		fbUnitTest.addString('<?xml version="1.0" ?>');
		fbUnitTest.addCrlf();

		fbUnitTest.addString('<testsuites>');
		fbUnitTest.addCrlf();

		pActTestSuite := getFirstTestSuite();

		WHILE (pActTestSuite <> 0) DO

			u16TestSuitIdx := u16TestSuitIdx+1;

			fbUnitTest.addString('<testsuite');
			fbUnitTest.addString(' name="');
			fbUnitTest.addString(pActTestSuite^.getId());
			fbUnitTest.addString('" tests="');
			u32Temp := pActTestSuite^.getNoOfTests();
			fbUnitTest.addValue(u32Temp);
			fbUnitTest.addString('" disabled="');
			u32Temp := 0;
			fbUnitTest.addValue(u32Temp);
			fbUnitTest.addString('" errors="');
			fbUnitTest.addValue(u32Temp);
			fbUnitTest.addString('" failures="');
			u32Temp := pActTestSuite^.getFailed();
			fbUnitTest.addValue(u32Temp);
			fbUnitTest.addString('" hostname="');
			fbUnitTest.addString('" id="');
			fbUnitTest.addvalue(u16TestSuitIdx);
			fbUnitTest.addString('" package="');
			fbUnitTest.addString(pActTestSuite^.getPath());
			fbUnitTest.addString('">');
			fbUnitTest.addCrlf();

			pTestCase := pActTestSuite^.getFirstTestCase();

			WHILE (pTestCase <> 0) DO

				fbUnitTest.addString('<testcase');
				fbUnitTest.addString(' name="');
				fbUnitTest.addString(pTestCase^.getId());
				fbUnitTest.addString('" assertions="');
				u32Temp := pTestCase^.getFailed() + pTestCase^.getPassed();
				fbUnitTest.addValue(u32Temp);
				fbUnitTest.addString('" classname="');
				fbUnitTest.addString(pTestCase^.getPath());
				fbUnitTest.addString(pTestCase^.getClassName());
				fbUnitTest.addString('" time="');
				u32Temp := pTestCase^.getTime();
				fbUnitTest.addTimeMs(u32Temp);
				fbUnitTest.addString('">');
				fbUnitTest.addCrlf();

				CASE pTestCase^.o_eResult OF

				EResult_t.eStatePassed :

					fbUnitTest.addString('<passed/>');

				EResult_t.eStateFailed, 
				EResult_t.eStateFailedFatal :
			
					fbUnitTest.addString('<failure');
					fbUnitTest.addString(' message="');
					fbUnitTest.addString(pTestCase^.getMessage());
					fbUnitTest.addString('"/>');
					
				EResult_t.eStateSkipped:

					fbUnitTest.addString('<skipped/>');

				END_CASE;
				
				fbUnitTest.addCrlf();	

				fbUnitTest.addString('</testcase>');
				fbUnitTest.addCrlf();		

				pTestCase := pActTestSuite^.getNextTestCase();
		
			END_WHILE

			fbUnitTest.addString('</testsuite>');
			fbUnitTest.addCrlf();	

			pActTestSuite := getNextTestSuite();

		END_WHILE

		fbUnitTest.addString('</testsuites>');
		fbUnitTest.addCrlf();

		u16ReportState := 22;

	22:
		IF fbUnitTest.o_bOpen  = TRUE AND 
		   fbUnitTest.o_bEmpty = TRUE THEN
			fbUnitTest.close();
		END_IF;

		IF fbUnitTest.o_bOpen  = FALSE THEN
			createReport 	:= ERetCode_t.eRetDone;
		END_IF;

// +++++++++++++++++++++++++++++++++++++++++++++++++++++++++++
//
//
// 
// +++++++++++++++++++++++++++++++++++++++++++++++++++++++++++
	100:

		IF pTestReport <> 0 THEN
			
			createReport := pTestReport^.create();		
			
		ELSE

			createReport := ERetCode_t.eRetDone;

		END_IF;

	ELSE
		createReport := ERetCode_t.eRetFailed;
	END_CASE;

	IF createReport = ERetCode_t.eRetDone THEN
		u16ReportState := 0;
	END_IF;
















(**)
END_METHOD

(******************************************************************************
Baustein: PRG_UnitTestLib.getFirstTestSuite
Spezifikation: doc/Spezifikation.pdf, Kap. x.y.z
-------------------------------------------------------------------------------
erstellt:
von:
Geändert:
von:
-------------------------------------------------------------------------------
Beschreibung
Diese Methode

-------------------------------------------------------------------------------
Input
-

Output
-
******************************************************************************)
{attribute 'hide'} 
METHOD PRIVATE getFirstTestSuite : TestSuiteHandle_t
VAR_INPUT
END_VAR

	u16Index := 0;
	getFirstTestSuite := a_pTestSuite[0];
END_METHOD

(******************************************************************************
Baustein: PRG_UnitTestLib.getNextTestSuite
Spezifikation: doc/Spezifikation.pdf, Kap. x.y.z
-------------------------------------------------------------------------------
erstellt:
von:
Geändert:
von:
-------------------------------------------------------------------------------
Beschreibung
Diese Methode

-------------------------------------------------------------------------------
Input
-

Output
-
******************************************************************************)
{attribute 'hide'} 
METHOD PRIVATE getNextTestSuite : TestSuiteHandle_t
VAR_INPUT
END_VAR

	getNextTestSuite := 0;
	u16Index 		 := u16Index + 1;

	IF u16Index < u16TestSuites THEN
		getNextTestSuite := a_pTestSuite[u16Index];
	END_IF;
END_METHOD

(******************************************************************************
Baustein: PRG_UnitTestLib.getTime
Spezifikation: doc/Spezifikation.pdf, Kap. x.y.z
-------------------------------------------------------------------------------
erstellt:
von:
Geändert:
von:
-------------------------------------------------------------------------------
Beschreibung
Diese Methode

-------------------------------------------------------------------------------
Input
-

Output
-
******************************************************************************)
{attribute 'hide'} 
METHOD getTime : TimeStruct
VAR_INPUT
END_VAR
VAR
END_VAR

	getTime := fbSystemTime.systemTime;
END_METHOD

{attribute 'hide'} 
METHOD PUBLIC LineCovered : BOOL
VAR_INPUT
	u16Pou  : UINT;
	u16Line : UINT;
END_VAR

	LineCovered := TRUE;
	
	//IF o_eState = EState_t.eStatePrepare OR 
	//   o_eState = EState_t.eStateExecute OR 
	//   o_eState = EState_t.eStateCleanUp THEN

		IF (u16Pou  > 0 AND u16Pou  <= u32MaxPouIdx ) AND
           (u16Line > 0 AND u16Line <= u32MaxLineIdx) THEN

			IF u16Pou > sCodeCoverage.u16MaxPouIndex THEN
				sCodeCoverage.u16MaxPouIndex := u16Pou;
			END_IF;
			IF u16Line > sCodeCoverage.u16MaxLineIndex THEN
				sCodeCoverage.u16MaxLineIndex := u16Line;
			END_IF;
			
			IF sCodeCoverage.aPou[u16Pou][u16Line] < 255 THEN
				sCodeCoverage.aPou[u16Pou][u16Line] := sCodeCoverage.aPou[u16Pou][u16Line]+1;
			END_IF;
		END_IF;

	//END_IF;
END_METHOD

(******************************************************************************
Baustein: PRG_UnitTestLib.logError
Spezifikation: doc/Spezifikation.pdf, Kap. x.y.z
-------------------------------------------------------------------------------
erstellt:
von:
Geändert:
von:
-------------------------------------------------------------------------------
Beschreibung
Diese Methode

-------------------------------------------------------------------------------
Input
i_strMessage

Output
-
******************************************************************************)
{attribute 'hide'} 
METHOD PROTECTED logError : BOOL
VAR_INPUT
	i_strMessage : StrMessage_t;
END_VAR

	ADSLOGSTR(msgCtrlMask 	:= ADSLOG_MSGTYPE_ERROR , 
			  msgFmtStr 	:= i_strMessage, 
			  strArg 		:= '');
END_METHOD

(******************************************************************************
Baustein: PRG_UnitTestLib.logInfo
Spezifikation: doc/Spezifikation.pdf, Kap. x.y.z
-------------------------------------------------------------------------------
erstellt:
von:
Geändert:
von:
-------------------------------------------------------------------------------
Beschreibung
Diese Methode

-------------------------------------------------------------------------------
Input
i_strMessage

Output
-
******************************************************************************)
{attribute 'hide'} 
METHOD PUBLIC logInfo : BOOL
VAR_INPUT
	i_strMessage : StrMessage_t;
END_VAR

	ADSLOGSTR(msgCtrlMask 	:= ADSLOG_MSGTYPE_HINT , 
			  msgFmtStr 	:= i_strMessage, 
			  strArg 		:= '');
END_METHOD

END_PROGRAM

// Source/Report/FB_TextReport
FUNCTION_BLOCK FB_TextReport EXTENDS FB_TestReportBase
VAR_INPUT
END_VAR
VAR_OUTPUT
END_VAR
VAR
END_VAR

(******************************************************************************
Baustein: FB_TestReportBase.BuildFile
Spezifikation: doc/Spezifikation.pdf, Kap. x.y.z
-------------------------------------------------------------------------------
erstellt:
von:
Geändert:
von:
-------------------------------------------------------------------------------
Beschreibung
Diese Methode muss vom ableitenden Baustein überschrieben werden und
wird von der Basisklasse aus aufgerufen wenn der Report erstellt werden
soll.

-------------------------------------------------------------------------------
Input
-

Output
-
******************************************************************************)
METHOD PROTECTED BuildFile : ERetCode_t
VAR_INPUT
	i_u32Line : UDINT;
END_VAR

	BuildFile := ERetCode_t.eRetBusy;

	CASE i_u32Line OF

	0: addString('Test Report :');
	   addDate(getTime());
	   addString(' - ');
	   addTime(getTime());
	1: addString('++++++++++++++++++++++++++++++++++++++++++++++++++');
	2: //
	3: //

	4: addString('Asserts gesamt: ');
	   addValue(sStatistic.u32Asserts);

	5: addString('Asserts passed: ');
	   addValue(sStatistic.u32Passed);

	6: addString('Asserts failed: ');
	   addValue(sStatistic.u32Failed);

	7: //

	9:  addString('Ergebnis : ');
		IF sStatistic.u32Failed > 0 THEN
			addString('FAILED');
		ELSE
			addString('PASSED');
		END_IF;

	10: addString('++++++++++++++++++++++++++++++++++++++++++++++++++');
	
	99: BuildFile := ERetCode_t.eRetDone;

	END_CASE;
END_METHOD

(******************************************************************************
Baustein: FB_TestReportBase.getFileName
Spezifikation: doc/Spezifikation.pdf, Kap. x.y.z
-------------------------------------------------------------------------------
erstellt:
von:
Geändert:
von:
-------------------------------------------------------------------------------
Beschreibung
Diese Methode muss vom ableitenden Baustein überschrieben werden und
wird von der Basisklasse aus aufgerufen wenn der Report erstellt werden
soll.

-------------------------------------------------------------------------------
Input
-

Output
-
******************************************************************************)
METHOD PROTECTED getFileName : ERetCode_t
VAR_INPUT
	i_pFileName : NameHandle_t;
	i_pPath		: PathHandle_t;
END_VAR
VAR
	sTime : TIMESTRUCT;
END_VAR

	i_pFileName^ := 'Exp_';
	i_pPath^ 	 := 'C:\Users\Administrator\Desktop\TestResult\';

	sTime := getTime();

	i_pFileName^ := Concat(i_pFileName^, WORD_TO_STRING(sTime.wYear));
	i_pFileName^ := Concat(i_pFileName^, DWORD_TO_DECSTR(sTime.wMonth, 2));
	i_pFileName^ := Concat(i_pFileName^, DWORD_TO_DECSTR(sTime.wDay  , 2));
	i_pFileName^ := Concat(i_pFileName^, '_');
	i_pFileName^ := Concat(i_pFileName^, DWORD_TO_DECSTR(sTime.wHour  , 2));
	i_pFileName^ := Concat(i_pFileName^, DWORD_TO_DECSTR(sTime.wMinute, 2));
	i_pFileName^ := Concat(i_pFileName^, '.txt');
END_METHOD

END_FUNCTION_BLOCK

// Test/FB_Test_Base
FUNCTION_BLOCK FB_Test_Base EXTENDS FB_UnitTestBase
VAR_INPUT
END_VAR
VAR_OUTPUT
END_VAR
VAR
END_VAR

(******************************************************************************
Baustein: FB_Test_Base.cleanup
Spezifikation: doc/Spezifikation.pdf, Kap. x.y.z
-------------------------------------------------------------------------------
erstellt:
von:
Geändert:
von:
-------------------------------------------------------------------------------
Beschreibung
Diese Methode...

-------------------------------------------------------------------------------
Input
-

Output
-
******************************************************************************)
METHOD PUBLIC cleanup : BOOL
VAR_INPUT
END_VAR

	cleanup := true;
END_METHOD

(******************************************************************************
Baustein: FB_Test_Base.execute
Spezifikation: doc/Spezifikation.pdf, Kap. x.y.z
-------------------------------------------------------------------------------
erstellt:
von:
Geändert:
von:
-------------------------------------------------------------------------------
Beschreibung
Diese Methode...

-------------------------------------------------------------------------------
Input
-

Output
-
******************************************************************************)
METHOD PUBLIC execute : BOOL
VAR_INPUT
END_VAR
VAR
	bValue1   : ARRAY[0..10] OF BOOL;
	bValue2   : ARRAY[0..10] OF BOOL;
	s8Value1  : ARRAY[0..10] OF SINT;
	s8Value2  : ARRAY[0..10] OF SINT;
	u8Value1  : ARRAY[0..10] OF USINT;
	u8Value2  : ARRAY[0..10] OF USINT;	
	s16Value1 : ARRAY[0..10] OF INT;
	s16Value2 : ARRAY[0..10] OF INT;
	u16Value1 : ARRAY[0..10] OF UINT;
	u16Value2 : ARRAY[0..10] OF UINT;		
	s32Value1 : ARRAY[0..10] OF DINT;
	s32Value2 : ARRAY[0..10] OF DINT;
	u32Value1 : ARRAY[0..10] OF UDINT;
	u32Value2 : ARRAY[0..10] OF UDINT;	
	r32Value1 : ARRAY[0..10] OF REAL;
	r32Value2 : ARRAY[0..10] OF REAL;
	r64Value1 : ARRAY[0..10] OF LREAL;
	r64Value2 : ARRAY[0..10] OF LREAL;
	strValue1 : ARRAY[0..10] OF STRING;
	strValue2 : ARRAY[0..10] OF STRING;
END_VAR


	bValue1[0] := TRUE;
	bValue2[0] := TRUE;
	
	setMessage('Teste Datentyp BOOL');
	assertEQUAL(bValue1[0], bValue2[0]);
	
	setMessage('Teste Datentyp Array of BOOL');
	assertEQUAL(bValue1, bValue2);

(**********************************************) 
	
	s8Value1[0] := 32;
	s8Value2[0] := 32;
	
	setMessage('Teste Datentyp SINT');
	assertEQUAL(s8Value1[0], s8Value2[0]);

	setMessage('Teste Datentyp Array of SINT');
	assertEQUAL(s8Value1, s8Value2);
(**********************************************) 	

	u8Value1[0] := 34;
	u8Value2[0] := 34;
	
	setMessage('Teste Datentyp USINT');
	assertEQUAL(u8Value1[0], u8Value2[0]);

	setMessage('Teste Datentyp Array of USINT');
	assertEQUAL(u8Value1, u8Value2);
(**********************************************) 	
	
	s16Value1[0] := 1323;
	s16Value2[0] := 1323;
	
	setMessage('Teste Datentyp INT');
	assertEQUAL(s16Value1[0], s16Value2[0]);

	setMessage('Teste Datentyp Array of INT');
	assertEQUAL(s16Value1, s16Value2);
(**********************************************) 	

	u16Value1[0] := 3124;
	u16Value2[0] := 3124;
	
	setMessage('Teste Datentyp UINT');
	assertEQUAL(u16Value1[0] , u16Value2[0] );

	setMessage('Teste Datentyp Array of UINT');
	assertEQUAL(u16Value1 , u16Value2);
(**********************************************) 	

	s32Value1[0] := 1244;
	s32Value2[0] := 1244;
	
	setMessage('Teste Datentyp DINT');
	assertEQUAL(s32Value1[0], s32Value2[0]);

	setMessage('Teste Datentyp Array of DINT');
	assertEQUAL(s32Value1, s32Value2);
(**********************************************) 	

	u32Value1[0] := 4344;
	u32Value2[0] := 4344;
	
	setMessage('Teste Datentyp UDINT');
	assertEQUAL(u32Value1[0], u32Value2[0]);

	setMessage('Teste Datentyp Array of UDINT');
	assertEQUAL(u32Value1, u32Value2);
(**********************************************) 	

	r32Value1[0] := 133.53245;
	r32Value2[0] := 133.53245;
	
	setMessage('Teste Datentyp REAL');
	assertEQUAL(r32Value1[0], r32Value2[0]);

	setMessage('Teste Datentyp Array of REAL');
	assertEQUAL(r32Value1, r32Value2);
(**********************************************) 	

	r64Value1[0] := 1232.53325;
	r64Value2[0] := 1232.53325;

	setMessage('Teste Datentyp LREAL');
	assertEQUAL(r64Value1[0], r64Value2[0]);

	setMessage('Teste Datentyp Array of LREAL');
	assertEQUAL(r64Value1, r64Value2);

(**********************************************) 	

	strValue1[0] := 'Hallo Welt';
	strValue2[0] := 'Hallo Welt';

	setMessage('Teste Datentyp String ist gleich');
	assertStringEqual(ADR(strValue1[0]), ADR(strValue2[0]));

	//setMessage('Teste Datentyp Array of String ist gleich');
	//assertEQUAL(strValue1, strValue2);

	strValue1[0] := 'Hallo Well';
	strValue2[0] := 'Hallo Welt';
	
	setMessage('Teste Datentyp String ist ungleich');
	assertStringNotEqual(ADR(strValue1[0]), ADR(strValue2[0]));

	//setMessage('Teste Datentyp Array of String ist ungleich');
	//assertNotEQUAL(strValue1, strValue2);
	
(**********************************************) 	





	execute := TRUE;
END_METHOD

(******************************************************************************
Baustein: FB_Test_Base.prepare
Spezifikation: doc/Spezifikation.pdf, Kap. x.y.z
-------------------------------------------------------------------------------
erstellt:
von:
Geändert:
von:
-------------------------------------------------------------------------------
Beschreibung
Diese Methode...

-------------------------------------------------------------------------------
Input
-

Output
-
******************************************************************************)
METHOD PUBLIC prepare : BOOL
VAR_INPUT
END_VAR

	prepare := true;
END_METHOD

END_FUNCTION_BLOCK

// Test/FB_Test_Base_Delay
FUNCTION_BLOCK FB_Test_Base_Delay EXTENDS FB_UnitTestBase
VAR_INPUT
END_VAR
VAR_OUTPUT
END_VAR
VAR
	fbDelay : TON;
END_VAR

(******************************************************************************
Baustein: FB_Test_Base_Delay.cleanup
Spezifikation: doc/Spezifikation.pdf, Kap. x.y.z
-------------------------------------------------------------------------------
erstellt:
von:
Geändert:
von:
-------------------------------------------------------------------------------
Beschreibung
Diese Methode...

-------------------------------------------------------------------------------
Input
-

Output
-
******************************************************************************)
METHOD PUBLIC cleanup : BOOL
VAR_INPUT
END_VAR

	cleanup := TRUE;
	
	fbDelay(IN := false);
END_METHOD

(******************************************************************************
Baustein: FB_Test_Base_Delay.execute
Spezifikation: doc/Spezifikation.pdf, Kap. x.y.z
-------------------------------------------------------------------------------
erstellt:
von:
Geändert:
von:
-------------------------------------------------------------------------------
Beschreibung
Diese Methode...

-------------------------------------------------------------------------------
Input
-

Output
-
******************************************************************************)
METHOD PUBLIC execute : BOOL
VAR_INPUT
END_VAR
VAR
	bValue1  : BOOL;
	bValue2  : BOOL;
	s32Value1 : DINT;
	s32Value2 : DINT;
	r32Value1 : REAL;
	r32Value2 : REAL;
END_VAR

	fbDelay(PT := t#250ms);

	bValue1 := TRUE;
	bValue2 := TRUE;
	assertEQUAL(bValue1, bValue2);

	s32Value1 := 1593;
	s32Value2 := 1593;
	assertEQUAL(s32Value1, s32Value2);

	r32Value1 := 5345.53245;
	r32Value2 := 5345.53245;
	assertEQUAL(r32Value1, r32Value2);

	execute := fbDelay.Q;
END_METHOD

(******************************************************************************
Baustein: FB_Test_Base_Delay.prepare
Spezifikation: doc/Spezifikation.pdf, Kap. x.y.z
-------------------------------------------------------------------------------
erstellt:
von:
Geändert:
von:
-------------------------------------------------------------------------------
Beschreibung
Diese Methode...

-------------------------------------------------------------------------------
Input
-

Output
-
******************************************************************************)
METHOD PUBLIC prepare : BOOL
VAR_INPUT
END_VAR

	prepare := TRUE;
	
	fbDelay.IN := true;
END_METHOD

END_FUNCTION_BLOCK

// Test/FB_Test_Base_Not
FUNCTION_BLOCK FB_Test_Base_Not EXTENDS FB_UnitTestBase
VAR_INPUT
END_VAR
VAR_OUTPUT
END_VAR
VAR
END_VAR

(******************************************************************************
Baustein: FB_Test_Base_Not.cleanup
Spezifikation: doc/Spezifikation.pdf, Kap. x.y.z
-------------------------------------------------------------------------------
erstellt:
von:
Geändert:
von:
-------------------------------------------------------------------------------
Beschreibung
Diese Methode...

-------------------------------------------------------------------------------
Input
-

Output
-
******************************************************************************)
METHOD PUBLIC cleanup : BOOL
VAR_INPUT
END_VAR

	cleanup := true;
END_METHOD

(******************************************************************************
Baustein: FB_Test_Base_Not.execute
Spezifikation: doc/Spezifikation.pdf, Kap. x.y.z
-------------------------------------------------------------------------------
erstellt:
von:
Geändert:
von:
-------------------------------------------------------------------------------
Beschreibung
Diese Methode...

-------------------------------------------------------------------------------
Input
-

Output
-
******************************************************************************)
METHOD PUBLIC execute : BOOL
VAR_INPUT
END_VAR
VAR
	bValue1   : ARRAY[0..10] OF BOOL;
	bValue2   : ARRAY[0..10] OF BOOL;
	s8Value1  : ARRAY[0..10] OF SINT;
	s8Value2  : ARRAY[0..10] OF SINT;
	u8Value1  : ARRAY[0..10] OF USINT;
	u8Value2  : ARRAY[0..10] OF USINT;	
	s16Value1 : ARRAY[0..10] OF INT;
	s16Value2 : ARRAY[0..10] OF INT;
	u16Value1 : ARRAY[0..10] OF UINT;
	u16Value2 : ARRAY[0..10] OF UINT;		
	s32Value1 : ARRAY[0..10] OF DINT;
	s32Value2 : ARRAY[0..10] OF DINT;
	u32Value1 : ARRAY[0..10] OF UDINT;
	u32Value2 : ARRAY[0..10] OF UDINT;	
	r32Value1 : ARRAY[0..10] OF REAL;
	r32Value2 : ARRAY[0..10] OF REAL;
	r64Value1 : ARRAY[0..10] OF LREAL;
	r64Value2 : ARRAY[0..10] OF LREAL;
END_VAR


	bValue1[0] := FALSE;
	bValue2[0] := TRUE;
	
	setMessage('Teste Datentyp BOOL');
	assertNotEQUAL(bValue1[0], bValue2[0]);
	
	setMessage('Teste Datentyp Array of BOOL');
	assertNotEQUAL(bValue1, bValue2);

(**********************************************) 
	
	s8Value1[0] := 31;
	s8Value2[0] := 32;
	
	setMessage('Teste Datentyp SINT');
	assertNotEQUAL(s8Value1[0], s8Value2[0]);

	setMessage('Teste Datentyp Array SINT');
	assertNotEQUAL(s8Value1, s8Value2);
(**********************************************) 	

	u8Value1[0] := 1;
	u8Value2[0] := 34;
	
	setMessage('Teste Datentyp USINT');
	assertNotEQUAL(u8Value1[0], u8Value2[0]);

	setMessage('Teste Datentyp Array of USINT');
	assertNotEQUAL(u8Value1, u8Value2);
(**********************************************) 	
	
	s16Value1[0] := 1323;
	s16Value2[0] := 4324;
	
	setMessage('Teste Datentyp INT');
	assertNotEQUAL(s16Value1[0], s16Value2[0]);

	setMessage('Teste Datentyp Array of INT');
	assertNotEQUAL(s16Value1, s16Value2);
(**********************************************) 	

	u16Value1[0] := 3124;
	u16Value2[0] := 4232;
	
	setMessage('Teste Datentyp UINT');
	assertNotEQUAL(u16Value1[0] , u16Value2[0] );

	setMessage('Teste Datentyp Array of UINT');
	assertNotEQUAL(u16Value1 , u16Value2);
(**********************************************) 	

	s32Value1[0] := 1244;
	s32Value2[0] := 1593;
	
	setMessage('Teste Datentyp DINT');
	assertNotEQUAL(s32Value1[0], s32Value2[0]);

	setMessage('Teste Datentyp Array of DINT');
	assertNotEQUAL(s32Value1, s32Value2);
(**********************************************) 	

	u32Value1[0] := 4344;
	u32Value2[0] := 3424;
	
	setMessage('Teste Datentyp UDINT');
	assertNotEQUAL(u32Value1[0], u32Value2[0]);

	setMessage('Teste Datentyp Array of UDINT');
	assertNotEQUAL(u32Value1, u32Value2);
(**********************************************) 	

	r32Value1[0] := 133.53245;
	r32Value2[0] := 5345.53245;
	
	setMessage('Teste Datentyp REAL');
	assertNotEQUAL(r32Value1[0], r32Value2[0]);

	setMessage('Teste Datentyp Array of REAL');
	assertNotEQUAL(r32Value1, r32Value2);
(**********************************************) 	

	r64Value1[0] := 1232.53325;
	r64Value2[0] := 1345.53325;

	setMessage('Teste Datentyp LREAL');
	assertNotEQUAL(r64Value1[0], r64Value2[0]);

	setMessage('Teste Datentyp Array of LREAL');
	assertNotEQUAL(r64Value1, r64Value2);

(**********************************************) 		
	execute := TRUE;
END_METHOD

(******************************************************************************
Baustein: FB_Test_Base_Not.prepare
Spezifikation: doc/Spezifikation.pdf, Kap. x.y.z
-------------------------------------------------------------------------------
erstellt:
von:
Geändert:
von:
-------------------------------------------------------------------------------
Beschreibung
Diese Methode...

-------------------------------------------------------------------------------
Input
-

Output
-
******************************************************************************)
METHOD PUBLIC prepare : BOOL
VAR_INPUT
END_VAR

	prepare := true;
END_METHOD

END_FUNCTION_BLOCK

// Test/FB_Test_Base_Ptr
FUNCTION_BLOCK FB_Test_Base_Ptr EXTENDS FB_UnitTestBase
VAR_INPUT
END_VAR
VAR_OUTPUT
END_VAR
VAR
END_VAR

(******************************************************************************
Baustein: FB_Test_Base.cleanup
Spezifikation: doc/Spezifikation.pdf, Kap. x.y.z
-------------------------------------------------------------------------------
erstellt:
von:
Geändert:
von:
-------------------------------------------------------------------------------
Beschreibung
Diese Methode...

-------------------------------------------------------------------------------
Input
-

Output
-
******************************************************************************)
METHOD PUBLIC cleanup : BOOL
VAR_INPUT
END_VAR

	cleanup := true;
END_METHOD

(******************************************************************************
Baustein: FB_Test_Base.execute
Spezifikation: doc/Spezifikation.pdf, Kap. x.y.z
-------------------------------------------------------------------------------
erstellt:
von:
Geändert:
von:
-------------------------------------------------------------------------------
Beschreibung
Diese Methode...

-------------------------------------------------------------------------------
Input
-

Output
-
******************************************************************************)
METHOD PUBLIC execute : BOOL
VAR_INPUT
END_VAR
VAR
	bValue1   : ARRAY[0..10] OF BOOL;
	bValue2   : ARRAY[0..10] OF BOOL;
	s8Value1  : ARRAY[0..10] OF SINT;
	s8Value2  : ARRAY[0..10] OF SINT;
	u8Value1  : ARRAY[0..10] OF USINT;
	u8Value2  : ARRAY[0..10] OF USINT;	
	s16Value1 : ARRAY[0..10] OF INT;
	s16Value2 : ARRAY[0..10] OF INT;
	u16Value1 : ARRAY[0..10] OF UINT;
	u16Value2 : ARRAY[0..10] OF UINT;		
	s32Value1 : ARRAY[0..10] OF DINT;
	s32Value2 : ARRAY[0..10] OF DINT;
	u32Value1 : ARRAY[0..10] OF UDINT;
	u32Value2 : ARRAY[0..10] OF UDINT;	
	r32Value1 : ARRAY[0..10] OF REAL;
	r32Value2 : ARRAY[0..10] OF REAL;
	r64Value1 : ARRAY[0..10] OF LREAL;
	r64Value2 : ARRAY[0..10] OF LREAL;
END_VAR


	bValue1[0] := TRUE;
	bValue2[0] := TRUE;
	
	setMessage('Teste Pointer to BOOL equal');
	assertPtrEQUAL(ADR(bValue1[0]), ADR(bValue1[0]));
	
	setMessage('Teste Pointer to BOOL NOT equal');
	assertPtrNOTEQUAL(ADR(bValue1), ADR(bValue2));

(**********************************************) 
	
	s8Value1[0] := 32;
	s8Value2[0] := 32;
	
	setMessage('Teste Pointer to BOOL SINT equal');
	assertPtrEQUAL(ADR(s8Value1[0]), ADR(s8Value1[0]));

	setMessage('Teste Pointer to SINT not equal');
	assertPtrNOTEQUAL(ADR(s8Value1), ADR(s8Value2));
(**********************************************) 	

	u8Value1[0] := 34;
	u8Value2[0] := 34;
	
	setMessage('Teste Pointer to USINT equal');
	assertPtrEQUAL(ADR(u8Value1[0]), ADR(u8Value1[0]));

	setMessage('Teste Pointer to USINT not equal');
	assertPtrNOTEQUAL(ADR(u8Value1), ADR(u8Value2));
(**********************************************) 	
	
	s16Value1[0] := 1323;
	s16Value2[0] := 1323;
	
	setMessage('Teste Pointer to INT equal');
	assertPtrEQUAL(ADR(s16Value1[0]), ADR(s16Value1[0]));

	setMessage('Teste Pointer to INT not equal');
	assertPtrNOTEQUAL(ADR(s16Value1), ADR(s16Value2));
(**********************************************) 	

	u16Value1[0] := 3124;
	u16Value2[0] := 3124;
	
	setMessage('Teste Pointer to UINT equal');
	assertPtrEQUAL(ADR(u16Value1[0]) , ADR(u16Value1[0]) );

	setMessage('Teste Pointer to  UINT not equal');
	assertPtrNOTEQUAL(ADR(u16Value1) , ADR(u16Value2));
(**********************************************) 	

	s32Value1[0] := 1244;
	s32Value2[0] := 1244;
	
	setMessage('Teste Pointer to DINT equal');
	assertPtrEQUAL(ADR(s32Value1[0]), ADR(s32Value1[0]));

	setMessage('Teste Pointer to  DINT not equal');
	assertPtrNOTEQUAL(ADR(s32Value1), ADR(s32Value2));
(**********************************************) 	

	u32Value1[0] := 4344;
	u32Value2[0] := 4344;
	
	setMessage('Teste Pointer to UDINT equal');
	assertPtrEQUAL(ADR(u32Value1[0]), ADR(u32Value1[0]));

	setMessage('Teste Pointer to  UDINT not equal');
	assertPtrNOTEQUAL(ADR(u32Value1), ADR(u32Value2));
(**********************************************) 	

	r32Value1[0] := 133.53245;
	r32Value2[0] := 133.53245;
	
	setMessage('Teste Pointer to REAL equal');
	assertPtrEQUAL(ADR(r32Value1[0]), ADR(r32Value1[0]));

	setMessage('Teste Pointer to  REAL not equal');
	assertPtrNOTEQUAL(ADR(r32Value1), ADR(r32Value2));
(**********************************************) 	

	r64Value1[0] := 1232.53325;
	r64Value2[0] := 1232.53325;

	setMessage('Teste Pointer to LREAL equal');
	assertPtrEQUAL(ADR(r64Value1[0]), ADR(r64Value1[0]));

	setMessage('Teste Pointer to LREAL not equal');
	assertPtrNOTEQUAL(ADR(r64Value1), ADR(r64Value2));

(**********************************************)

	setMessage('Teste Pointer = 0');	
	assertPtrNull(pActual := 0);
	
	setMessage('Teste Pointer <> 0');	
	assertPtrNotNull(pActual := ADR(r32Value1[0]));	
	
(**********************************************)	
	
	
	
	
	
	
	
	
	
	execute := TRUE;
END_METHOD

(******************************************************************************
Baustein: FB_Test_Base.prepare
Spezifikation: doc/Spezifikation.pdf, Kap. x.y.z
-------------------------------------------------------------------------------
erstellt:
von:
Geändert:
von:
-------------------------------------------------------------------------------
Beschreibung
Diese Methode...

-------------------------------------------------------------------------------
Input
-

Output
-
******************************************************************************)
METHOD PUBLIC prepare : BOOL
VAR_INPUT
END_VAR

	prepare := true;
END_METHOD

END_FUNCTION_BLOCK
